// TwinCAT 3 PLC project Plc
// ProgramVersion: 3.1.4023.0
// libraries:
//   Tc2_Standard, * (Beckhoff Automation GmbH)
//   Tc2_System, * (Beckhoff Automation GmbH)
//   Tc3_Module, * (Beckhoff Automation GmbH)
// project tree:
//   / PlcTask.TcTTO (not stored)
//   DUTs/IO/PDOs/ InfoData_6F19DB2B.TcDUT (not stored), Channel_42CA91F7.TcDUT, WcState_0B2B16F9.TcDUT, InfoData_E68C61CD.TcDUT (not stored), InfoData_2A97D6CF.TcDUT (not stored), Inputs_A65FACA4.TcDUT (not stored), Outputs_23C0ED1D.TcDUT (not stored)
//   DUTs/IO/Boxes/ EK1100_1FC0878B.TcDUT (not stored), EL2809_2B6483BD.TcDUT
//   DUTs/IO/Devices/ SyncUnitTask_2D604ED5.TcDUT (not stored), SyncUnitTasks_6FEB8257.TcDUT (not stored), SyncUnits_99E584AF.TcDUT (not stored)
//   DUTs/IO/Topology/ Term_1_EK1100_DD7D5547.TcDUT (not stored), Device_1_EtherCAT_DDCD551C.TcDUT (not stored)
//   DUTs/IO/Base/ EtcSlaveBase_82538BE2.TcDUT (not stored), EtcSlaveBase_82538BE2.TcDUT (not stored), EtcSlaveBase_82538BE2.TcDUT (not stored), EtcSlaveTerminalBase_947E5A46.TcDUT (not stored), EtcSlaveBoxBase_77A0E4A7.TcDUT (not stored), EtcSlaveEndTerminalBase_866C7F0C.TcDUT (not stored), InputBase_8311D824.TcDUT (not stored), OutputBase_10CEE7DE.TcDUT (not stored), EtcMasterBase_62654B43.TcDUT (not stored)
//   GVLs/ GVL_iXlinker.TcGVL (not stored)
// real-time tasks:
//   TASK PlcTask: cycle T#10ms, priority 20, ADS port 350
// I/O:
//   DEVICE Device 1 (EtherCAT), AmsNetId 172.20.30.238.2.1
//     Term 1 (EK1100) [EK1100 EtherCAT Coupler (2A E-Bus)]
//       Term 2 (EL2809) [EL2809 16Ch. Dig. Output 24V, 0.5A]
// variable links:
//   Plc/Plc Instance <-> Device 1 (EtherCAT)/Term 1 (EK1100)
//     PlcTask Inputs/GVL_iXlinker.Device_1_EtherCAT.Term_1_EK1100.InfoData.State <-> InfoData/State
//   Plc/Plc Instance <-> Device 1 (EtherCAT)/Term 1 (EK1100)/Term 2 (EL2809)
//     PlcTask Outputs/GVL_iXlinker.Device_1_EtherCAT.Term_1_EK1100.Term_2_EL2809.Channel_{1..16}.Output <-> Channel {1..16}/Output  (16 links)
//     PlcTask Inputs/GVL_iXlinker.Device_1_EtherCAT.Term_1_EK1100.Term_2_EL2809.WcState.WcState <-> WcState/WcState
//     PlcTask Inputs/GVL_iXlinker.Device_1_EtherCAT.Term_1_EK1100.Term_2_EL2809.InfoData.State <-> InfoData/State
//   Plc/Plc Instance <-> Device 1 (EtherCAT)
//     PlcTask Inputs/GVL_iXlinker.Device_1_EtherCAT.SyncUnits._default._unreferenced.WcState.WcState <-> SyncUnits/<default>/<unreferenced>/WcState/WcState
//     PlcTask Inputs/GVL_iXlinker.Device_1_EtherCAT.SyncUnits._default._unreferenced.InfoData.ObjectId <-> SyncUnits/<default>/<unreferenced>/InfoData/ObjectId
//     PlcTask Inputs/GVL_iXlinker.Device_1_EtherCAT.SyncUnits._default._unreferenced.InfoData.State <-> SyncUnits/<default>/<unreferenced>/InfoData/State
//     PlcTask Inputs/GVL_iXlinker.Device_1_EtherCAT.SyncUnits._default._unreferenced.InfoData.SlaveCount <-> SyncUnits/<default>/<unreferenced>/InfoData/SlaveCount
//     PlcTask Inputs/GVL_iXlinker.Device_1_EtherCAT.SyncUnits._default.PlcTask.WcState.WcState <-> SyncUnits/<default>/PlcTask/WcState/WcState
//     PlcTask Inputs/GVL_iXlinker.Device_1_EtherCAT.SyncUnits._default.PlcTask.InfoData.ObjectId <-> SyncUnits/<default>/PlcTask/InfoData/ObjectId
//     PlcTask Inputs/GVL_iXlinker.Device_1_EtherCAT.SyncUnits._default.PlcTask.InfoData.State <-> SyncUnits/<default>/PlcTask/InfoData/State
//     PlcTask Inputs/GVL_iXlinker.Device_1_EtherCAT.SyncUnits._default.PlcTask.InfoData.SlaveCount <-> SyncUnits/<default>/PlcTask/InfoData/SlaveCount
//     PlcTask Inputs/GVL_iXlinker.Device_1_EtherCAT.Inputs.SlaveCount <-> Inputs/SlaveCount
//     PlcTask Inputs/GVL_iXlinker.Device_1_EtherCAT.Inputs.DevState <-> Inputs/DevState
//     PlcTask Inputs/GVL_iXlinker.Device_1_EtherCAT.Inputs.Frm0State <-> Inputs/Frm0State
//     PlcTask Inputs/GVL_iXlinker.Device_1_EtherCAT.Inputs.Frm0WcState <-> Inputs/Frm0WcState
//     PlcTask Inputs/GVL_iXlinker.Device_1_EtherCAT.Inputs.Frm0InputToggle <-> Inputs/Frm0InputToggle
//     PlcTask Outputs/GVL_iXlinker.Device_1_EtherCAT.Outputs.DevCtrl <-> Outputs/DevCtrl
//     PlcTask Outputs/GVL_iXlinker.Device_1_EtherCAT.Outputs.Frm0Ctrl <-> Outputs/Frm0Ctrl
//     PlcTask Outputs/GVL_iXlinker.Device_1_EtherCAT.Outputs.Frm0WcCtrl <-> Outputs/Frm0WcCtrl
//     PlcTask Inputs/GVL_iXlinker.Device_1_EtherCAT.InfoData.ChangeCount <-> InfoData/ChangeCount
//     PlcTask Inputs/GVL_iXlinker.Device_1_EtherCAT.InfoData.DevId <-> InfoData/DevId
//     PlcTask Inputs/GVL_iXlinker.Device_1_EtherCAT.InfoData.AmsNetId <-> InfoData/AmsNetId
//     PlcTask Inputs/GVL_iXlinker.Device_1_EtherCAT.InfoData.CfgSlaveCount <-> InfoData/CfgSlaveCount
//     PlcTask Inputs/GVL_iXlinker.Device_1_EtherCAT.InfoData.DcToTcTimeOffset <-> InfoData/DcToTcTimeOffset
//     PlcTask Inputs/GVL_iXlinker.Device_1_EtherCAT.InfoData.DcToExtTimeOffset <-> InfoData/DcToExtTimeOffset

// ---- DUTs/IO/PDOs/Channel_42CA91F7.TcDUT
{attribute 'GeneratedUsingTerminal: EL2809-0000-0018'}
{attribute addProperty BoxType "EL2809-0000-0018"}
{attribute addProperty Id "OutputAT %Q*BOOL1"}
{attribute addProperty CRC "1120571895"}
{attribute addProperty Size "1"}
TYPE Channel_42CA91F7 EXTENDS OutputBase_10CEE7DE :
STRUCT
	{attribute addProperty Name "Output"}
	Output AT %Q* : BOOL;
END_STRUCT
END_TYPE

// ---- DUTs/IO/PDOs/WcState_0B2B16F9.TcDUT
{attribute 'GeneratedUsingTerminal: EL2809-0000-0018'}
{attribute addProperty BoxType "EL2809-0000-0018"}
{attribute addProperty Id "WcStateAT %I*BOOL1"}
{attribute addProperty CRC "187373305"}
{attribute addProperty Size "1"}
TYPE WcState_0B2B16F9 :
STRUCT
	{attribute addProperty Name "WcState"}
	WcState AT %I* : BOOL;
END_STRUCT
END_TYPE

// ---- DUTs/IO/Boxes/EL2809_2B6483BD.TcDUT
{attribute 'GeneratedUsingTerminal: EL2809-0000-0018'}
{attribute addProperty BoxType "EL2809-0000-0018"}
{attribute addProperty Description "EL2809 16Ch. Dig. Output 24V, 0.5A"}
{attribute addProperty Physics "KK"}
{attribute addProperty Id "Channel_1AT %Q*Channel_42CA91F71Channel_2AT %Q*Channel_42CA91F71Channel_3AT %Q*Channel_42CA91F71Channel_4AT %Q*Channel_42CA91F71Channel_5AT %Q*Channel_42CA91F71Channel_6AT %Q*Channel_42CA91F71Channel_7AT %Q*Channel_42CA91F71Channel_8AT %Q*Channel_42CA91F71Channel_9AT %Q*Channel_42CA91F71Channel_10AT %Q*Channel_42CA91F71Channel_11AT %Q*Channel_42CA91F71Channel_12AT %Q*Channel_42CA91F71Channel_13AT %Q*Channel_42CA91F71Channel_14AT %Q*Channel_42CA91F71Channel_15AT %Q*Channel_42CA91F71Channel_16AT %Q*Channel_42CA91F71WcStateAT %I*WcState_0B2B16F91InfoDataAT %I*InfoData_6F19DB2B2"}
{attribute addProperty CRC "728007613"}
{attribute addProperty Size "19"}
TYPE EL2809_2B6483BD EXTENDS EtcSlaveTerminalBase_947E5A46 :
STRUCT
	{attribute addProperty Name "Channel_1"}
	Channel_1 : Channel_42CA91F7;
	{attribute addProperty Name "Channel_2"}
	Channel_2 : Channel_42CA91F7;
	{attribute addProperty Name "Channel_3"}
	Channel_3 : Channel_42CA91F7;
	{attribute addProperty Name "Channel_4"}
	Channel_4 : Channel_42CA91F7;
	{attribute addProperty Name "Channel_5"}
	Channel_5 : Channel_42CA91F7;
	{attribute addProperty Name "Channel_6"}
	Channel_6 : Channel_42CA91F7;
	{attribute addProperty Name "Channel_7"}
	Channel_7 : Channel_42CA91F7;
	{attribute addProperty Name "Channel_8"}
	Channel_8 : Channel_42CA91F7;
	{attribute addProperty Name "Channel_9"}
	Channel_9 : Channel_42CA91F7;
	{attribute addProperty Name "Channel_10"}
	Channel_10 : Channel_42CA91F7;
	{attribute addProperty Name "Channel_11"}
	Channel_11 : Channel_42CA91F7;
	{attribute addProperty Name "Channel_12"}
	Channel_12 : Channel_42CA91F7;
	{attribute addProperty Name "Channel_13"}
	Channel_13 : Channel_42CA91F7;
	{attribute addProperty Name "Channel_14"}
	Channel_14 : Channel_42CA91F7;
	{attribute addProperty Name "Channel_15"}
	Channel_15 : Channel_42CA91F7;
	{attribute addProperty Name "Channel_16"}
	Channel_16 : Channel_42CA91F7;
	{attribute addProperty Name "WcState"}
	WcState : WcState_0B2B16F9;
	{attribute addProperty Name "InfoData"}
	InfoData : InfoData_6F19DB2B;
END_STRUCT
END_TYPE
